KUKA KRL program: St1_Test_Mill.src, St1_Test_Mill.dat

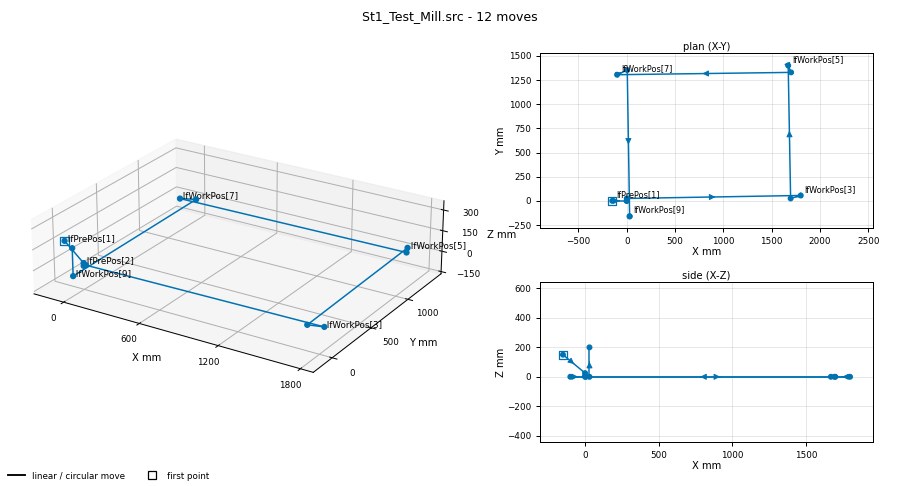
[picture p0: tool path of St1_Test_Mill.src, 12 of 15 moves have a stored position in this frame; points joined in program order, loops and branches not executed]
--- St1_Test_Mill.src ---
&ACCESS RVEO
&REL 5
DEF  St1_Test_Mill (lnActSt :IN)
   INT lnActSt,lnUsedBase,lnUsedTool
   INT lnJobNr


   ;FOLD INIT
      CONTINUE
      IF ($T1 OR $T2)THEN
         GLOBAL INTERRUPT DECL 3 WHEN $STOPMESS==TRUE DO IR_STOPM ( )
         INTERRUPT ON 3
         BAS (#INITMOV,0)
         lnActSt = 2
         PTP $POS_ACT
      ENDIF

      PTP XHOME

     ; Used Base and tool
      lnUsedBase = 11
      lnUsedTool = 11
      gnLastToolNr = 3


      gfMillingOffset = $NULLFRAME
      gfMillingOffset.Z = -(grCuttingDepth*(gnMillingCounter-1))

      BASE_DATA[lnUsedBase] = BASE_DATA[16]:gfBaseShift[lnActSt];:gfMillingOffset
      TOOL_DATA[lnUsedTool] = TOOL_DATA[4] :{X 0,Y 0,Z 0,A 0,B 0,C 0}
      grUsedRPM = GetMillingRPM(grTool_VC[gnLastToolNr], grTool_Diameter[gnLastToolNr])
      grUsedMillingSpeed = GetMillingSpeed(grUsedRPM, grTool_ToothCount[gnLastToolNr], grTool_FeedPerTooth[gnLastToolNr])
   ;ENDFOLD
   ;MoveSettings (nBase: IN, nTool: IN, nAcc: IN, nVel : IN )


   SpindleRun(grUsedRPM,#CLOCKWISE)
   WAIT SEC 10

   MoveSettings(lnUsedBase, lnUsedTool, 100, 500)
   PTP lfPrePos[1] C_PTP
   MoveSettings(lnUsedBase, lnUsedTool, 100, 200)
   LIN lfPrePos[2] C_DIS


   MoveSettings(lnUsedBase, lnUsedTool, 100, grUsedMillingSpeed)
   LIN lfWorkPos[1] C_DIS

   LIN lfWorkPos[2]

   LIN lfWorkPos[3]

   LIN lfWorkPos[4]

   LIN lfWorkPos[5]

   LIN lfWorkPos[6]

   LIN lfWorkPos[7]

   LIN lfWorkPos[8]

   LIN lfWorkPos[9]


   MoveSettings(lnUsedBase, lnUsedTool, 100, 20)

   WAIT SEC 0

   SpindleStop( )
   LIN lfWorkPos[10]

   WAIT SEC 0

  MoveSettings(lnUsedBase, lnUsedTool, 100, 2000)

   PTP XHOME





END

DEF endOfJob()
   gbJob1StartedSt[1] = FALSE
   gbJob1DoneSt[1]    = TRUE
   gnMillingCounter = gnMillingCounter+1
END

--- St1_Test_Mill.dat ---
&ACCESS RVEO
&REL 5
DEFDAT  St1_Test_Mill


DECL FRAME lfPrePos[3]
lfPrePos[1]={X -150.000,Y 0.0,Z 150.000,A 0.0,B 0.0,C 0.0}
lfPrePos[2]={X 0.0,Y 0.0,Z 25.0,A 0.0,B 0.0,C 0.0}
lfPrePos[3]={X 0.0,Y 0.0,Z 0.0,A 0.0,B 0.0,C 0.0}


DECL FRAME lfWorkPos[12]
   lfWorkPos[1]={X 0,Y 0,Z 5.000,A 0.0,B 0.0,C 0.0}
   lfWorkPos[2]={X 0,Y 25.0,Z 0.0000,A 0.0,B 0.0,C 0.0}

   lfWorkPos[3]={X 1800,Y 56.0,Z 0.0000,A -73.0,B 0.0,C 0.0}
   lfWorkPos[4]={X 1695,Y 25.0,Z 0.0000,A -73.0,B 0.0,C 0.0}
   lfWorkPos[5]={X 1670,Y 1400.0,Z 0.0000,A 15.0,B 0.0,C 0.0}
   lfWorkPos[6]={X 1700,Y 1329.0,Z 0.0000,A 15.0,B 0.0,C 0.0}
   lfWorkPos[7]={X -100,Y 1305.0,Z 0.0000,A -15.0,B 0.0,C 0.0}
   lfWorkPos[8]={X 5.3,Y 1353,Z 0.0000,A -15.0,B 0.0,C 0.0}
   lfWorkPos[9]={X 30,Y -160.0,Z 0.0000,A 63.0, B 0.0,C 0.0}
   lfWorkPos[10]={X 30,Y -160.0,Z 200.0000,A 0, B 0.0,C 0.0}


   lfWorkPos[11]={X 0,Y 0.0,Z 0.0000,A 0.0,B 0.0,C 0.0}
   lfWorkPos[12]={X 0,Y 0.0,Z 0.0000,A 0.0,B 0.0,C 0.0}


ENDDAT
